(* PLC project E-motor.project, CODESYS CODESYS V3.5 SP10 *)
(* stored: creationDateTime 2018-02-26T10:15:15.1331641, modificationDateTime 2018-02-26T10:14:57.7045276 *)

PROGRAM Main
  VAR_INPUT
    START : BOOL;
    TZ : BOOL;
  END_VAR
  VAR
    T1 : TON;
    T2 : TON;
    RS1 : RS;
    RS2 : RS;
    RT1 : R_TRIG;
  END_VAR
  VAR_OUTPUT
    ZZ : BOOL;
    FZ : BOOL;
  END_VAR

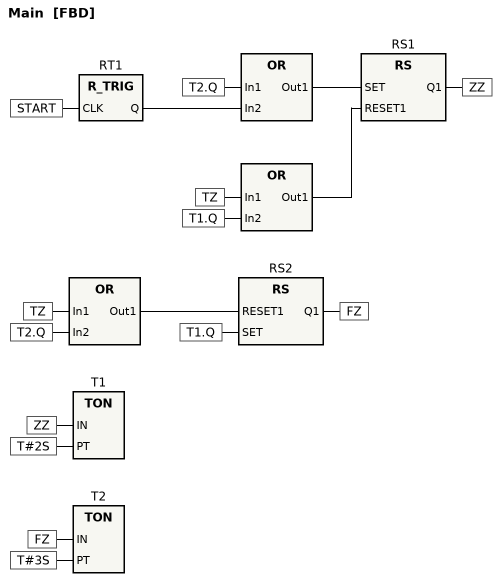
(* FBD diagram, written out as Structured Text *)
RT1(CLK := START);
RS1(SET := T2.Q OR RT1.Q, RESET1 := TZ OR T1.Q);
ZZ := RS1.Q1;
RS2(RESET1 := TZ OR T2.Q, SET := T1.Q);
FZ := RS2.Q1;
T1(IN := ZZ, PT := T#2S);
T2(IN := FZ, PT := T#3S);
END_PROGRAM

CONFIGURATION Application
  RESOURCE Application ON PLC
    TASK Task(INTERVAL := T#1000ms, PRIORITY := 1);
    PROGRAM Main WITH Task : Main;
  END_RESOURCE
END_CONFIGURATION
